// Mitsubishi GX Works2 project: clock   PLC: Q02/Q02H
// clock

PROGRAM MAIN
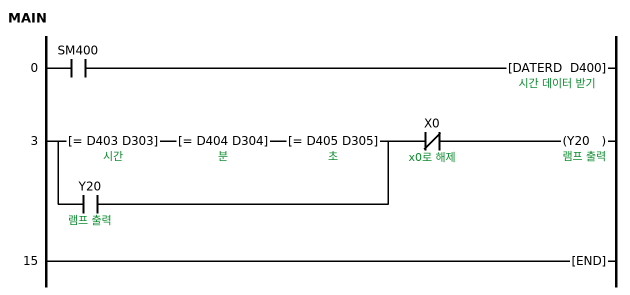
0     LD      SM400
      DATERD  D400  ; 시간 데이터 받기
3     LD=     D403 D303  ; 시간
      AND=    D404 D304  ; 분
      AND=    D405 D305  ; 초
      OR      Y20  ; 램프 출력
      ANI     X0  ; x0로 해제
      OUT     Y20  ; 램프 출력
15    END
END_PROGRAM
